// TIA Portal V16 export
// export: Created 2022-07-21T09:35:20.188693Z, ExportSetting WithDefaults, DisplayName Totally Integrated Automation Portal, DisplayVersion V16 Update 4, DisplayName TIA Portal Version Control Interface, DisplayVersion V16 Update 2, DisplayName TIA Portal Openness, DisplayVersion V16 Update 4, DisplayName SINAMICS Startdrive Advanced, DisplayVersion V16 Update 5, DisplayName SINAMICS Startdrive G130, G150, S120, S150, SINAMICS MV, S210, DisplayVersion V16 Update 5, DisplayName SINAMICS Startdrive G110M, G120, G120C, G120D, G120P, G115D, DisplayVersion V16 Update 5, DisplayName STEP 7 Professional, DisplayVersion V16 Update 4, DisplayName STEP 7 Safety, DisplayVersion V16, DisplayName WinCC Advanced, DisplayVersion V16 Update 4
DATA_BLOCK "idbCoolingHandling"   // DB13
VERSION : 0.1
// stored: AutoNumber true, DBAccessibleFromOPCUA true, InstanceOfName fbCoolingHandling, InstanceOfType FB
"fbCoolingHandling"
   // VAR_INPUT
   //    inNewFilterIN : Bool;
   //    inNewFilterOUT : Bool;
   //    inEmptyingLineRequest : Bool;
   //    inSlotSensors : "typeCoolingSensorSlot";
   //    inGateClose : Bool;
   //    inGroup : "typeGroup";
   // END_VAR
   // VAR_OUTPUT
   //    ouCoolingEmpty : Bool;
   //    ouFillingActive : Bool;
   //    ouEmptyingActive : Bool;
   //    ouCountOccupiedSlots : Int;
   //    ouCountBlockedSlots : Int;
   //    ouEnableEntranceForRobot : Bool;
   //    ouLevelForRobot : Int;
   //    ouTypeProgram : Int;
   //    ouMoveTTPermitt : Bool;
   //    ouError : Bool;
   //    ouStatus : Word;
   // END_VAR
   // VAR_IN_OUT
   //    ioPlus1Pos : Bool;
   //    ioPlus2Pos : Bool;
   //    ioData : "typeCoolingTracking";
   //    ioSensors : Array[*] of Bool;
   //    ioDrive : "typeRotaryDrive";
   // END_VAR
   // VAR
   //    sError : Word;
   //    sTriggerIN : R_TRIG;
   //    sTriggerOUT : R_TRIG;
   // END_VAR
   // VAR RETAIN
   //    sAvaLevelTab : Array[1.."Cooling_Max_Level"] of Bool;
   //    sAvaLevelNo : Int;
   //    sAvaLevelStart : Int;
   // END_VAR
   // VAR
   //    sGetTime : "fbGetTimeStruct";
   //    sDate : "typeDateSplit";
   //    sDateArray : Array[0..2] of String[4];
   //    sCharArray : Array[0..20] of Char;
   //    sStr : String;
   //    sDaTLastEntrance : Date_And_Time;
   // END_VAR
   // VAR RETAIN
   //    sStoreSlotNo : Int;
   //    sAvaStoreSlotNo : Bool;
   // END_VAR
BEGIN
END_DATA_BLOCK
